INTERFACE I_STRING EXTENDS I_Datatype

PROPERTY PUBLIC Value : REFERENCE TO T_MaxString
GET
END_GET
END_PROPERTY

END_INTERFACE

(* stored: Version 1.1.0.1, ProductVersion 3.1.4024.15
   Itf I_STRING: Id {24a8d6a5-a43e-0403-286c-5609f9ee3852}
   Property Value: Id {9ce269e8-b3fe-0b8a-02fb-4ec8ece58e11}
   Get Get: Id {be9f4e24-4ae9-0303-0d86-8eb0c99cd5f4} *)
